(* CODESYS project BagCountController.xml

Project tree, tasks and I/O mapping:
  function block BagCountController [CFC]
*)

// BagCountController
FUNCTION_BLOCK BagCountController
VAR_INPUT
	BagOpenFail: BOOL;
	BagOpenFailReset: BOOL;
	BagFailure: BOOL;
	MaxBagOpenFails: UINT;
	MaxBagFails: UINT;
END_VAR
VAR_OUTPUT
	BagFail: BOOL;
	BagOpenFailCount: UINT;
	BagFailCount: UINT;
	BagAdvanceAlarm: BOOL;
END_VAR
VAR
	_BagOpenFailureCounter: CTU;
END_VAR

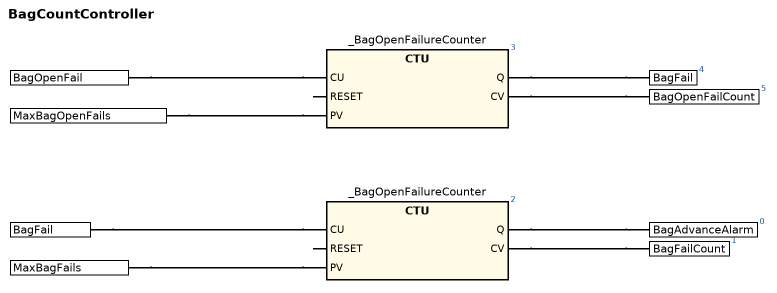
BagAdvanceAlarm := _BagOpenFailureCounter.Q;
BagFailCount := _BagOpenFailureCounter.CV;
_BagOpenFailureCounter(CU := BagFail, PV := MaxBagFails); // CTU
_BagOpenFailureCounter(CU := BagOpenFail, PV := MaxBagOpenFails); // CTU
BagFail := _BagOpenFailureCounter.Q;
BagOpenFailCount := _BagOpenFailureCounter.CV;

END_FUNCTION_BLOCK
